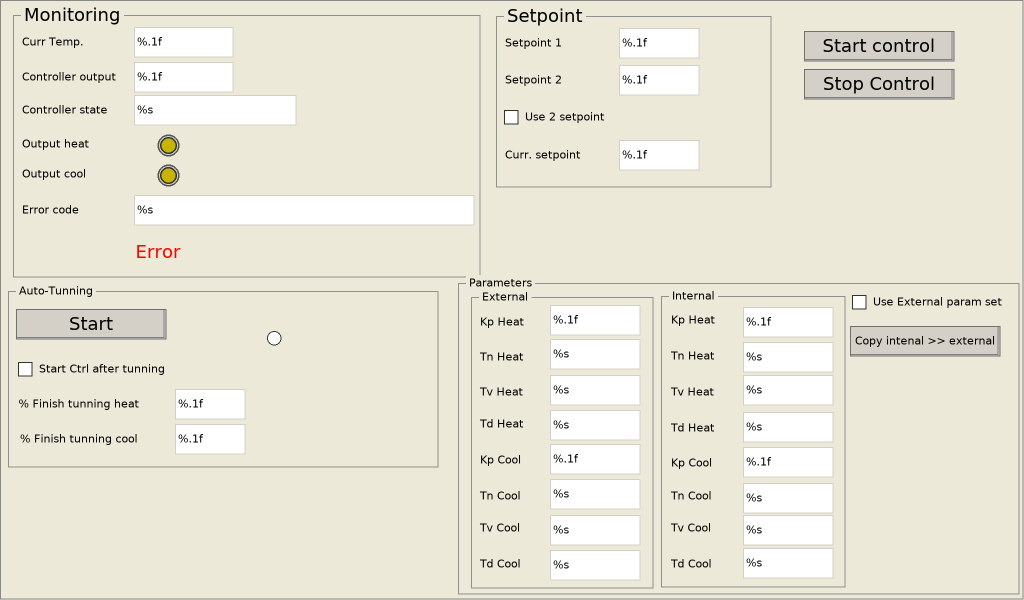
VISUALIZATION Visualization  // 1024x600
    GroupBox (496,8 275x179), "Setpoint"
        Checkbox (6,94 120x30), "Use 2 setpoint", variable: MAIN.bSelSetpoint
        Textfield (123,20 80x30), "%.1f", text variable: MAIN.tempSetpoint[1]
            OnMouseClick: write the text variable via Default
        Textfield (123,57 80x30), "%.1f", text variable: MAIN.tempSetpoint[2]
            OnMouseClick: write the text variable via Default
        Label (6,57 110x30), "Setpoint 2"
        Label (6,20 110x30), "Setpoint 1"
        Textfield (123,132 80x30), "%.1f", text variable: MAIN.activeSetpoint
        Label (6,132 110x30), "Curr. setpoint"
    GroupBox (13,7 467x270), "Monitoring"
        Textfield (121,20 99x30), "%.1f", text variable: MAIN.currTemp
        Textfield (121,88 162x30), "%s", text variable: MAIN.eCtrlState
        Label (6,88 110x30), "Controller state"
        Label (6,20 110x30), "Curr Temp."
        Textfield (121,55 99x30), "%.1f", text variable: MAIN.fyAnalogOutput
        Label (6,55 110x30), "Controller output"
        Label (6,122 160x30), "Output heat"
        Lamp1 (143,126 25x25), variable: MAIN.bOutputHeat, style: Lamp-Lamp1-Yellow
        Label (6,152 160x30), "Output cool"
        Textfield (121,188 340x30), "%s", text variable: MAIN.errId
        Label (93,230 104x30), "Error", invisible if: not MAIN.bBlinkError
    GroupBox (458,275 561x319), "Parameters"
        GroupBox (13,14 182x299), "External"
            Label (6,18 70x30), "Kp Heat"
            Label (6,53 70x30), "Tn Heat"
            Label (6,88 70x30), "Tv Heat"
            Label (6,120 70x30), "Td Heat"
            Label (6,156 70x30), "Kp Cool"
            Label (6,192 70x30), "Tn Cool"
            Label (6,224 70x30), "Tv Cool"
            Label (6,260 70x30), "Td Cool"
            Textfield (79,16 90x30), "%.1f", text variable: MAIN.externalParams.KpHeat
            Textfield (79,50 90x30), "%s", text variable: MAIN.externalParams.TnHeat
            Textfield (79,86 90x30), "%s", text variable: MAIN.externalParams.TvHeat
            Textfield (79,121 90x30), "%s", text variable: MAIN.externalParams.TdHeat
            Textfield (79,155 90x30), "%.1f", text variable: MAIN.externalParams.KpCool
            Textfield (79,190 90x30), "%s", text variable: MAIN.externalParams.TnCool
            Textfield (79,226 90x30), "%s", text variable: MAIN.externalParams.TvCool
            Textfield (79,261 90x30), "%s", text variable: MAIN.externalParams.TdCool
        GroupBox (203,13 184x299), "Internal"
            Label (7,17 70x30), "Kp Heat"
            Label (7,53 70x30), "Tn Heat"
            Label (7,89 70x30), "Tv Heat"
            Label (7,125 70x30), "Td Heat"
            Label (7,160 70x30), "Kp Cool"
            Label (7,193 70x30), "Tn Cool"
            Label (7,225 70x30), "Tv Cool"
            Label (7,261 70x30), "Td Cool"
            Textfield (82,19 90x30), "%.1f", text variable: MAIN.internalParams.KpHeat
            Textfield (82,54 90x30), "%s", text variable: MAIN.internalParams.TnHeat
            Textfield (82,87 90x30), "%s", text variable: MAIN.internalParams.TvHeat
            Textfield (82,124 90x30), "%s", text variable: MAIN.internalParams.TdHeat
            Textfield (82,159 90x30), "%.1f", text variable: MAIN.internalParams.KpCool
            Textfield (82,195 90x30), "%s", text variable: MAIN.internalParams.TnCool
            Textfield (82,227 90x30), "%s", text variable: MAIN.internalParams.TvCool
            Textfield (82,260 90x30), "%s", text variable: MAIN.internalParams.TdCool
        Checkbox (392,12 172x30), "Use External param set", tooltip "When activated select the external params", variable: MAIN.stControllerParameter.bSelCtrlParameterSet
        Button (392,51 150x30), "Copy intenal >> external"
            tap MAIN.bCopyParams
    GroupBox (8,283 430x184), "Auto-Tunning"
        Button (8,26 150x30), "Start"
            tap MAIN.startAutoTunning
        Checkbox (8,71 163x30), "Start Ctrl after tunning", variable: MAIN.bStartCtrlAfterTunning
        Textfield (167,106 70x30), "%.1f", text variable: MAIN.stControllerParameter.fEndTunePercentHeating
            OnMouseClick: write the text variable via Default, min 10, max 90
        Label (6,106 130x30), "% Finish tunning heat"
        Textfield (167,141 70x30), "%.1f", text variable: MAIN.stControllerParameter.fEndTunePercentCooling
            OnMouseClick: write the text variable via Default, min 10, max 90
        RadioButton (257,8 169x94), variable: MAIN.iTunningType
            Areas[0]: Text=Tunning fast
            Areas[1]: Text=Tunning medium
            Areas[2]: Text=Tunning no overshoot
    Lamp1 (156,163 25x25), variable: MAIN.bOutputCool, style: Lamp-Lamp1-Yellow
    Label (19,195 104x30), "Error code"
    Label (14,424 130x30), "% Finish tunning cool"
    Button (804,31 150x30), "Start control"
        tap MAIN.startController
    Button (804,69 150x30), "Stop Control"
        tap MAIN.stopController
END_VISUALIZATION

(* stored: Version 1.1.0.1, ProductVersion 3.1.4024.12
   Visu Visualization: Id {84a3e8b4-b9e8-4cde-8e24-1d375dafd015} *)
